// TIA Portal V17 export
// export: Created 2023-12-22T15:08:10.1349876Z, ExportSetting WithDefaults, DisplayName Totally Integrated Automation Portal, DisplayVersion V17, DisplayName TIA Portal Openness, DisplayVersion V17, DisplayName TIA Portal Version Control Interface, DisplayVersion V17, DisplayName STEP 7 Professional, DisplayVersion V17, DisplayName STEP 7 Safety, DisplayVersion V17, DisplayName WinCC Advanced, DisplayVersion V17
DATA_BLOCK "PS_Main_DB"   // DB10
VERSION : 0.1
// stored: AutoNumber false, DBAccessibleFromOPCUA true, DBAccessibleFromWebserver true, InstanceOfName PS_Main, InstanceOfType FB
"PS_Main"
   // VAR_IN_OUT
   //    PS_REQ : Int;
   //    PS_cnt : Int;
   // END_VAR
   // VAR RETAIN
   //    Step_Up { S7_SetPoint := 'True'} : Array[1..6] of Real;
   //    Step_Down { S7_SetPoint := 'True'} : Array[1..6] of Real;
   //    PS_One { S7_SetPoint := 'True'} : Array[0..10] of "PS_One";
   //    PS_All { S7_SetPoint := 'True'} : Int := 7;
   //    PS_Group { S7_SetPoint := 'True'} : Int := 5;
   //    PS_Reserv { S7_SetPoint := 'True'} : Int := 2;
   //    PS_Ready : Int;
   //    PS_CMD : Int;
   //    PS_Work : Int;
   //    PS_Load : Int;
   //    PS_SP_Hz : Real;
   //    PS_Point : Real;
   //    PS_min_cnt : Int;
   // END_VAR
BEGIN
   Step_Up[1] := 0.5;   // Быстрый разгон
   Step_Up[2] := 0.5;   // Плавный разгон
   Step_Up[3] := 0.5;   // Рабочая точка
   Step_Up[4] := 0.05;   // Плавное замедление
   Step_Up[5] := 0.05;   // Быстрое замделение
   Step_Up[6] := 0.05;
   Step_Down[1] := 0.025;   // Быстрый разгон
   Step_Down[2] := 0.025;   // Плавный разгон
   Step_Down[3] := 0.5;   // Рабочая точка
   Step_Down[4] := 0.5;   // Плавное замедление
   Step_Down[5] := 0.5;   // Быстрое замделение
   Step_Down[6] := 0.5;
   PS_One[0..10].Min := FALSE;
   PS_One[0].T_Delay.SP_M := 10;
   PS_One[1..7].T_Delay.SP_M := 1;
   PS_One[8..10].T_Delay.SP_M := 10;
   PS_One[0..10].T_Delay.SP_S := 0;
   PS_One[0..10].T_PE_Delay.SP_M := 0;
   PS_One[0..10].T_PE_Delay.SP_S := 30;
END_DATA_BLOCK
